PROGRAM P_Demo_FB_DMXGetSlotInfo
VAR
    fbGetSlotInfo     : FB_DMXGetSlotInfo;            // 读各槽功能信息
    stDmxCmdBuffer    : ST_DMXCommandBuffer;          // 与通讯 FB 共用
    wTargetManufId    : WORD := 16#4241;              // 目标灯具厂商 ID
    dwTargetDeviceId  : DWORD := 16#12131415;         // 目标灯具设备 ID
    byTargetPort      : BYTE := 0;                    // 根设备通道 0
    bDoRead           : BOOL := FALSE;                // 在线给一次上升沿触发
    bBusy             : BOOL;
    bError            : BOOL;
    udiErrId          : UDINT;
    arrSlotInfo       : ARRAY [0..45] OF ST_DMXSlotInfo;  // 各槽功能信息(最多 46)
END_VAR

// ============================================================
// Tc2_DMX.FB_DMXGetSlotInfo 演示程序
// ============================================================
// 场景：自动构建通道映射表：一次读出某灯所有槽功能类型，PLC 据此自动关联各 DMX 通道到控制变量。
// 价值：一次调用拿到全部槽功能，自动化通道映射，比逐槽 FB_DMXGetSlotDescription 更快建立对应关系。
// 验证：给 bDoRead 一次上升沿 -> bBusy 短暂 TRUE -> 回 FALSE 后 arrSlotInfo[0..] 含设备各槽功能类型（占用 N 个槽则前 N 项有效）。
// 验证步骤：
//   1. 右键 PLC 项目下 POUs 文件夹 → Add → Existing Item → 选本 .TcPOU 文件
//   2. 引用 Tc2_DMX；同项目里放一个 FB_EL6851CommunicationEx 实例并共用 stDmxCmdBuffer（非 CycleMode）
//   3. 编译 → 登录 → 运行；按上方『验证』行在线给上升沿观察
// ============================================================

fbGetSlotInfo(
    bStart                     := bDoRead,
    wDestinationManufacturerId := wTargetManufId,
    dwDestinationDeviceId      := dwTargetDeviceId,
    byPortId                   := byTargetPort,
    dwOptions                  := 0,
    stCommandBuffer            := stDmxCmdBuffer,
    bBusy                      => bBusy,
    bError                     => bError,
    udiErrorId                 => udiErrId,
    arrSlotInfos               => arrSlotInfo
);

END_PROGRAM

(* stored: Version 1.1.0.1, ProductVersion 3.1.4024.5
   POU P_Demo_FB_DMXGetSlotInfo: Id {4ce59bae-5938-53cc-b081-029648a7466f}, SpecialFunc None *)
